PROGRAM TestRunner
VAR
    EventTests        : TEventTests;
    HandlerList_Tests : THandlerList_Tests;
    ExecutionTests    : TExecutionTests;
    Test_LicenceCheck : TTest_LicenceCheck;
END_VAR

TcUnit.RUN();

END_PROGRAM

(* stored: Version 1.1.0.1, ProductVersion 3.1.4024.3
   POU TestRunner: Id {05f63fc0-82d5-4467-8277-011f38ba0570}, SpecialFunc None *)
